// TIA Portal V17 export
// export: Created 2021-12-03T08:13:10.6546653Z, ExportSetting WithDefaults, DisplayName Totally Integrated Automation Portal, DisplayVersion V17, DisplayName TIA Portal Openness, DisplayVersion V17, DisplayName TIA Portal Version Control Interface, DisplayVersion V17, DisplayName STEP 7 Professional, DisplayVersion V17, DisplayName STEP 7 Safety, DisplayVersion V17, DisplayName WinCC Advanced, DisplayVersion V17
FUNCTION_BLOCK "FFB_EmStpButton"   // FB200, F_FBD
VERSION : 0.1
// stored: AutoNumber false, IsIECCheckEnabled false, UDAEnableTagReadback false
   VAR
      P1 { S7_SetPoint := 'True'} : ESTOP1;
      P2 { S7_SetPoint := 'True'} : ESTOP1;
      P3 { S7_SetPoint := 'True'} : ESTOP1;
      AccCons { S7_SetPoint := 'True'} : ESTOP1;
      Dosimetr { S7_SetPoint := 'True'} : ESTOP1;
   END_VAR
BEGIN

REGION Network 1: Em Stp P1
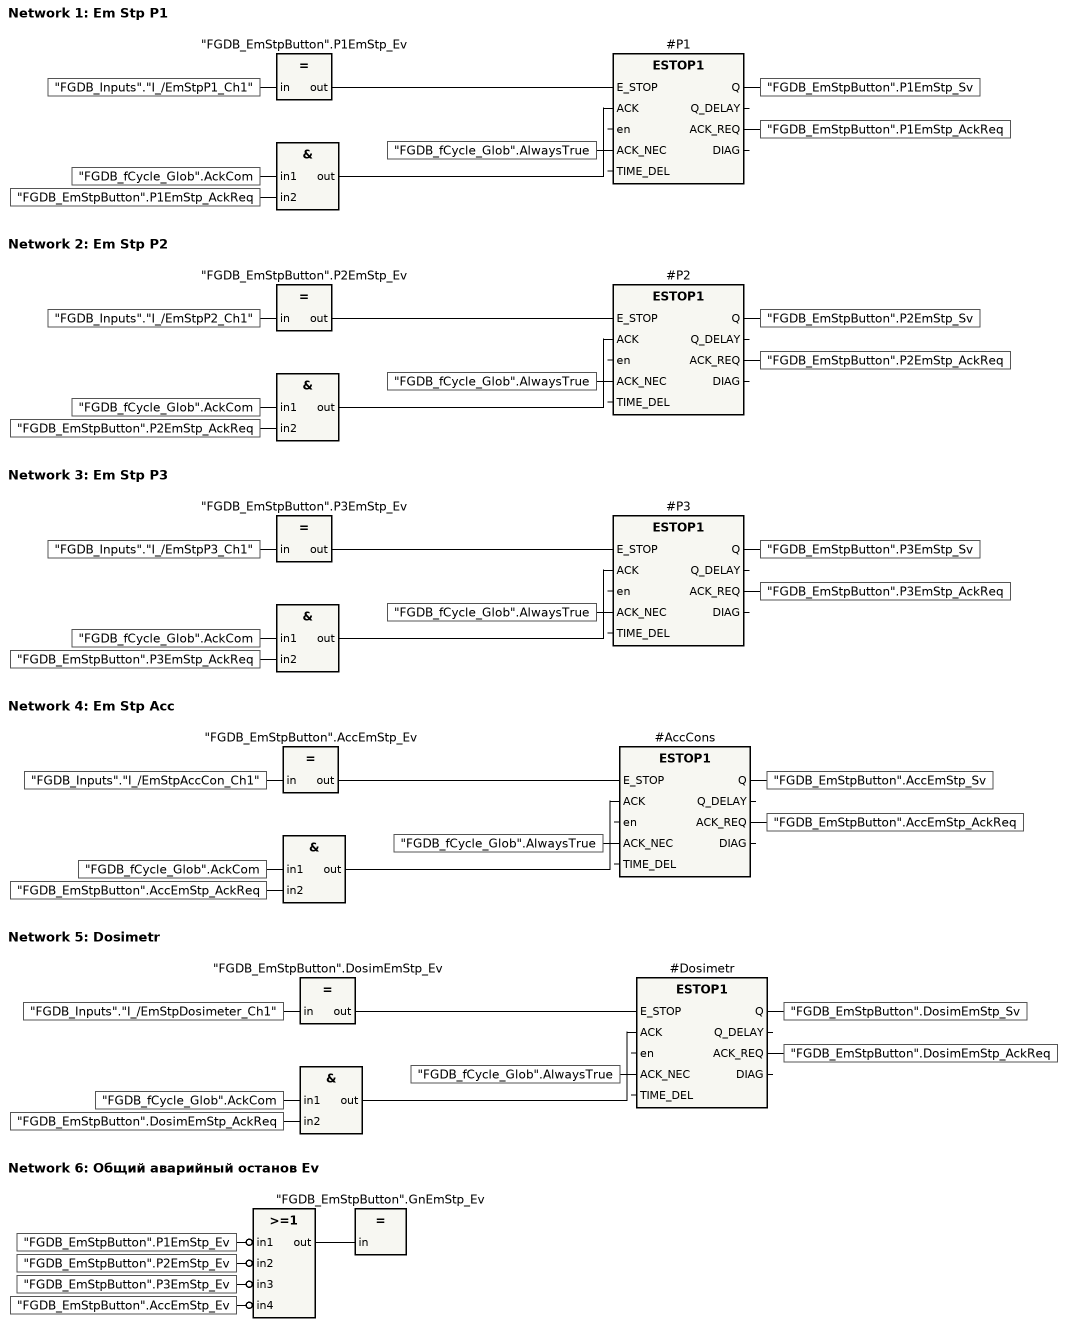
   "FGDB_EmStpButton".P1EmStp_Ev := "FGDB_Inputs"."I_/EmStpP1_Ch1";
   #P1(E_STOP := "FGDB_Inputs"."I_/EmStpP1_Ch1",   // ESTOP1
       ACK := "FGDB_fCycle_Glob".AckCom AND "FGDB_EmStpButton".P1EmStp_AckReq,
       ACK_NEC := "FGDB_fCycle_Glob".AlwaysTrue,
       Q => "FGDB_EmStpButton".P1EmStp_Sv,
       ACK_REQ => "FGDB_EmStpButton".P1EmStp_AckReq);
END_REGION

REGION Network 2: Em Stp P2
   "FGDB_EmStpButton".P2EmStp_Ev := "FGDB_Inputs"."I_/EmStpP2_Ch1";
   #P2(E_STOP := "FGDB_Inputs"."I_/EmStpP2_Ch1",   // ESTOP1
       ACK := "FGDB_fCycle_Glob".AckCom AND "FGDB_EmStpButton".P2EmStp_AckReq,
       ACK_NEC := "FGDB_fCycle_Glob".AlwaysTrue,
       Q => "FGDB_EmStpButton".P2EmStp_Sv,
       ACK_REQ => "FGDB_EmStpButton".P2EmStp_AckReq);
END_REGION

REGION Network 3: Em Stp P3
   "FGDB_EmStpButton".P3EmStp_Ev := "FGDB_Inputs"."I_/EmStpP3_Ch1";
   #P3(E_STOP := "FGDB_Inputs"."I_/EmStpP3_Ch1",   // ESTOP1
       ACK := "FGDB_fCycle_Glob".AckCom AND "FGDB_EmStpButton".P3EmStp_AckReq,
       ACK_NEC := "FGDB_fCycle_Glob".AlwaysTrue,
       Q => "FGDB_EmStpButton".P3EmStp_Sv,
       ACK_REQ => "FGDB_EmStpButton".P3EmStp_AckReq);
END_REGION

REGION Network 4: Em Stp Acc
   "FGDB_EmStpButton".AccEmStp_Ev := "FGDB_Inputs"."I_/EmStpAccCon_Ch1";
   #AccCons(E_STOP := "FGDB_Inputs"."I_/EmStpAccCon_Ch1",   // ESTOP1
            ACK := "FGDB_fCycle_Glob".AckCom AND "FGDB_EmStpButton".AccEmStp_AckReq,
            ACK_NEC := "FGDB_fCycle_Glob".AlwaysTrue,
            Q => "FGDB_EmStpButton".AccEmStp_Sv,
            ACK_REQ => "FGDB_EmStpButton".AccEmStp_AckReq);
END_REGION

REGION Network 5: Dosimetr
   "FGDB_EmStpButton".DosimEmStp_Ev := "FGDB_Inputs"."I_/EmStpDosimeter_Ch1";
   #Dosimetr(E_STOP := "FGDB_Inputs"."I_/EmStpDosimeter_Ch1",   // ESTOP1
             ACK := "FGDB_fCycle_Glob".AckCom AND "FGDB_EmStpButton".DosimEmStp_AckReq,
             ACK_NEC := "FGDB_fCycle_Glob".AlwaysTrue,
             Q => "FGDB_EmStpButton".DosimEmStp_Sv,
             ACK_REQ => "FGDB_EmStpButton".DosimEmStp_AckReq);
END_REGION

REGION Network 6: Общий аварийный останов Ev
   "FGDB_EmStpButton".GnEmStp_Ev := NOT "FGDB_EmStpButton".P1EmStp_Ev OR NOT "FGDB_EmStpButton".P2EmStp_Ev OR NOT "FGDB_EmStpButton".P3EmStp_Ev OR NOT "FGDB_EmStpButton".AccEmStp_Ev;
END_REGION

REGION Network 7: Общий аварийный останов AckRq
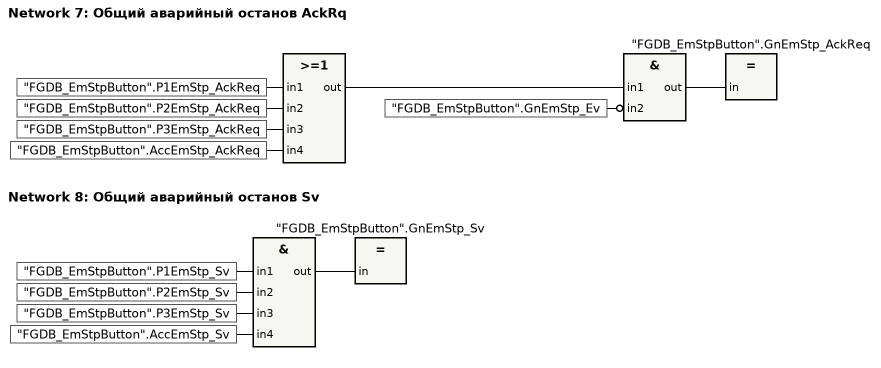
   "FGDB_EmStpButton".GnEmStp_AckReq := ("FGDB_EmStpButton".P1EmStp_AckReq OR "FGDB_EmStpButton".P2EmStp_AckReq OR "FGDB_EmStpButton".P3EmStp_AckReq OR "FGDB_EmStpButton".AccEmStp_AckReq) AND NOT "FGDB_EmStpButton".GnEmStp_Ev;
END_REGION

REGION Network 8: Общий аварийный останов Sv
   "FGDB_EmStpButton".GnEmStp_Sv := "FGDB_EmStpButton".P1EmStp_Sv AND "FGDB_EmStpButton".P2EmStp_Sv AND "FGDB_EmStpButton".P3EmStp_Sv AND "FGDB_EmStpButton".AccEmStp_Sv;
END_REGION
END_FUNCTION_BLOCK
